// TIA Portal V20 export
TYPE "LGM_LKinCtrl_ControlNodeMonitoring"
// stored: Access Published
   STRUCT
      groupPower : Struct
         busy { ExternalWritable := 'False'} : Bool;   // TRUE: FB is not finished and new output values can be expected
         error { ExternalWritable := 'False'} : Bool;   // TRUE: An error occurred during the execution of the FB
         axesEnabled { ExternalWritable := 'False'} : Bool := FALSE;   // TRUE: all axes of axesGroup enabled; FALSE: all axes of axesGroup disabled
         diagnostics { ExternalWritable := 'False'} : "LKinCtrl_typeAuxFCDiagnostics";   // Diagnostics information of FB (optional)
      END_STRUCT;
      groupHome : Struct
         done { ExternalWritable := 'False'} : Bool;   // axesGroup successfully referenced
         busy { ExternalWritable := 'False'} : Bool;   // FB is not finished and new output values can be expected
         active { ExternalWritable := 'False'} : Bool;   // FB in control of axesGroup / kinematic in motion
         commandAborted { ExternalWritable := 'False'} : Bool;   // command is aborted by another command
         error { ExternalWritable := 'False'} : Bool;   // an error occurred during the execution of the FB
         diagnostics { ExternalWritable := 'False'} : "LKinCtrl_typeAuxFCDiagnostics";   // diagnostics information of FB (optional)
      END_STRUCT;
      groupReset : Struct
         done { ExternalWritable := 'False'} : Bool;   // axesGroup successfully referenced
         busy { ExternalWritable := 'False'} : Bool;   // FB is not finished and new output values can be expected
         active { ExternalWritable := 'False'} : Bool;   // FB in control of axesGroup / kinematic in motion
         commandAborted { ExternalWritable := 'False'} : Bool;   // command is aborted by another command
         error { ExternalWritable := 'False'} : Bool;   // an error occurred during the execution of the FB
         diagnostics { ExternalWritable := 'False'} : "LKinCtrl_typeAuxFCDiagnostics";   // diagnostics information of FB (optional)
      END_STRUCT;
      movePath : Struct
         done { ExternalAccessible := 'False'; ExternalVisible := 'False'; ExternalWritable := 'False'} : Bool;
         busy { ExternalWritable := 'False'} : Bool;   // TRUE: FB is not finished and new output values can be expected
         active { ExternalWritable := 'False'} : Bool;   // FB in control of axesGroup / kinematic in motion
         commandAborted { ExternalAccessible := 'False'; ExternalVisible := 'False'; ExternalWritable := 'False'} : Bool;
         error { ExternalAccessible := 'False'; ExternalVisible := 'False'; ExternalWritable := 'False'} : Bool;
         status { ExternalWritable := 'False'} : Word := 0;   // status of the FB
         diagnostics { ExternalWritable := 'False'} : "LKinCtrl_typeMovePathDiagnostics";   // diagnostics information of FB
         activePathData { ExternalWritable := 'False'} : String["LKINCTRL_LENGTH_OF_PATHDATA_NAME"];   // name of actual PathData
         activeCmdNo { ExternalAccessible := 'False'; ExternalVisible := 'False'; ExternalWritable := 'False'} : DInt;
         remainingDistanceActCmd { ExternalAccessible := 'False'; ExternalVisible := 'False'; ExternalWritable := 'False'} : LReal;
         readyForNextPath { ExternalAccessible := 'False'; ExternalVisible := 'False'; ExternalWritable := 'False'} : Bool;
         activeUserFrames { ExternalWritable := 'False'} : Array["LKINCTRL_CS_NO_OF_FIRST_USER_FRAME".."LKINCTRL_CS_NO_OF_LAST_USER_FRAME"] of "LKinCtrl_typeFrame";   // Currently acitve user frames
         selectedPath { ExternalAccessible := 'False'; ExternalVisible := 'False'; ExternalWritable := 'False'} : DInt;
      END_STRUCT;
      hmiLogic : Struct
         editor : Struct
            busy : Bool;   // TRUE: FB is not finished and new output values can be expected
            valid : Bool;   // TRUE: FB outputs are valid
            status : Word := 0;   // 16#0000 - 16#7FFF: Status of the FB, 16#8000 - 16#FFFF: Error identification
            enableInfeed : Bool;   // TRUE: Enable infeed, FALSE: Disable infeed.
            enableAxesCoupling : Bool;   // TRUE: Enable axes coupling of kinematics axes, FALSE: Disable axes coupling. Defined in settings.
            acknowledgeInfeed : Bool;   // Rising edge: Acknowledge infeed.
            selectedPathNumber : DInt;   // Currently selected path number in editor.
         END_STRUCT;
         diagnostics : Struct
            busy : Bool;   // TRUE: FB is not finished and new output values can be expected
            valid : Bool;   // TRUE: FB outputs are valid
            status : Word := 0;   // 16#0000 - 16#7FFF: Status of the FB, 16#8000 - 16#FFFF: Error identification
         END_STRUCT;
      END_STRUCT;
   END_STRUCT;
   // groupPower.diagnostics.status := 0;
END_TYPE
